FUNCTION_BLOCK TelemetryUnpack (* Telemetry_CAT helper: unpacks the TelemetryConfig struct into MQTT_CONNECTION scalar inputs (whole-struct in + ST member access — no struct-member connections, which EAE rejects) *)
  (* Standard: 61499-2 *)
  (* Version 0.1, 6/22/2026, easensoy, WMG, Config:TelemetryConfig -> QI/ConnectionID/URL/ClientIdentifier/ValidateCert/CACert scalars *)
  PACKAGE Main;
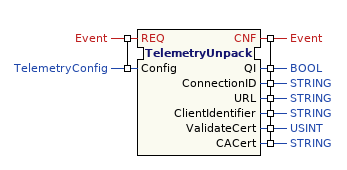
  EVENT_INPUT
    REQ WITH Config; (* Unpack request *)
  END_EVENT
  EVENT_OUTPUT
    CNF WITH QI, ConnectionID, URL, ClientIdentifier, ValidateCert, CACert; (* Unpack confirm *)
  END_EVENT
  VAR_INPUT
    Config : TelemetryConfig; (* Resource telemetry connection config *)
  END_VAR
  VAR_OUTPUT
    QI : BOOL;
    ConnectionID : STRING;
    URL : STRING;
    ClientIdentifier : STRING;
    ValidateCert : USINT;
    CACert : STRING;
  END_VAR
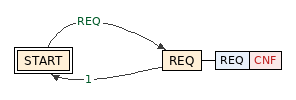
  EC_STATES
    START; (* Initial State *)
    REQ : REQ -> CNF; (* Unpack *)
  END_STATES
  EC_TRANSITIONS
    START TO REQ := REQ;
    REQ TO START := 1;
  END_TRANSITIONS
  ALGORITHM REQ IN ST: (* Copy each Config struct member to its scalar output *)
QI := Config.QI;
ConnectionID := Config.ConnectionID;
URL := Config.URL;
ClientIdentifier := Config.ClientIdentifier;
ValidateCert := Config.ValidateCert;
CACert := Config.CACert;
  END_ALGORITHM
END_FUNCTION_BLOCK
